PROGRAM Axis03_Command
VAR
//System_Bit
	Always_ON	:	BOOL	:=TRUE	;//상시 ON 
	Always_OFF	:	BOOL	:=FALSE	;//상시 OFF

//Motor_Command
	Axis03: AXIS_REF;											//Y축
	Axis03_MC_Power: MC_Power;
	Axis03_MC_Home: FB_HomeBeforeMoveAX8000;
	Axis03_Jog: MC_Jog;	
	Axis03_Home_Pos_Move: MC_MoveAbsolute;
	Axis03_Wait_Pos_Move: MC_MoveAbsolute;
	Axis03_Target_Pos_Move: MC_MoveAbsolute;
	Axis03_Work_End_Move: MC_MoveAbsolute;
	Axis03_Maint_Move: MC_MoveAbsolute;
	Axis03_Tool_Change: MC_MoveAbsolute;	
	Axis03_Calibration: MC_MoveAbsolute;	

	Timer02: TON;
END_VAR
VAR // added by the converter: edge detectors and wires of the graphical bodies
    _rt1, _rt2, _rt3 : R_TRIG;
END_VAR

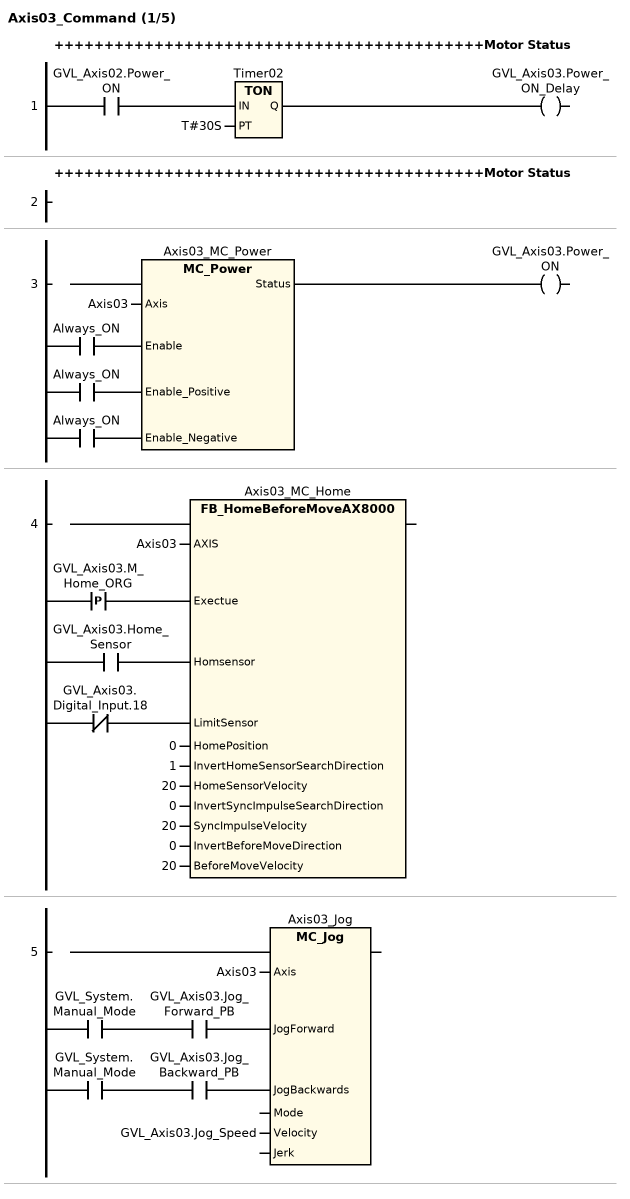
// NETWORK 1: +++++++++++++++++++++++++++++++++++++++++++Motor Status
Timer02(IN := GVL_Axis02.Power_ON, PT := T#30S); // TON
GVL_Axis03.Power_ON_Delay := Timer02.Q;

// NETWORK 2: +++++++++++++++++++++++++++++++++++++++++++Motor Status

// NETWORK 3
Axis03_MC_Power(
    Axis := Axis03,
    Enable := Always_ON,
    Enable_Positive := Always_ON,
    Enable_Negative := Always_ON); // MC_Power
GVL_Axis03.Power_ON := Axis03_MC_Power.Status;

// NETWORK 4
_rt1(CLK := GVL_Axis03.M_Home_ORG);
Axis03_MC_Home(
    AXIS := Axis03,
    Exectue := _rt1.Q,
    Homsensor := GVL_Axis03.Home_Sensor,
    LimitSensor := NOT GVL_Axis03.Digital_Input.18,
    HomePosition := 0,
    InvertHomeSensorSearchDirection := 1,
    HomeSensorVelocity := 20,
    InvertSyncImpulseSearchDirection := 0,
    SyncImpulseVelocity := 20,
    InvertBeforeMoveDirection := 0,
    BeforeMoveVelocity := 20); // FB_HomeBeforeMoveAX8000

// NETWORK 5
Axis03_Jog(
    Axis := Axis03,
    JogForward := GVL_System.Manual_Mode AND GVL_Axis03.Jog_Forward_PB,
    JogBackwards := GVL_System.Manual_Mode AND GVL_Axis03.Jog_Backward_PB,
    Velocity := GVL_Axis03.Jog_Speed); // MC_Jog

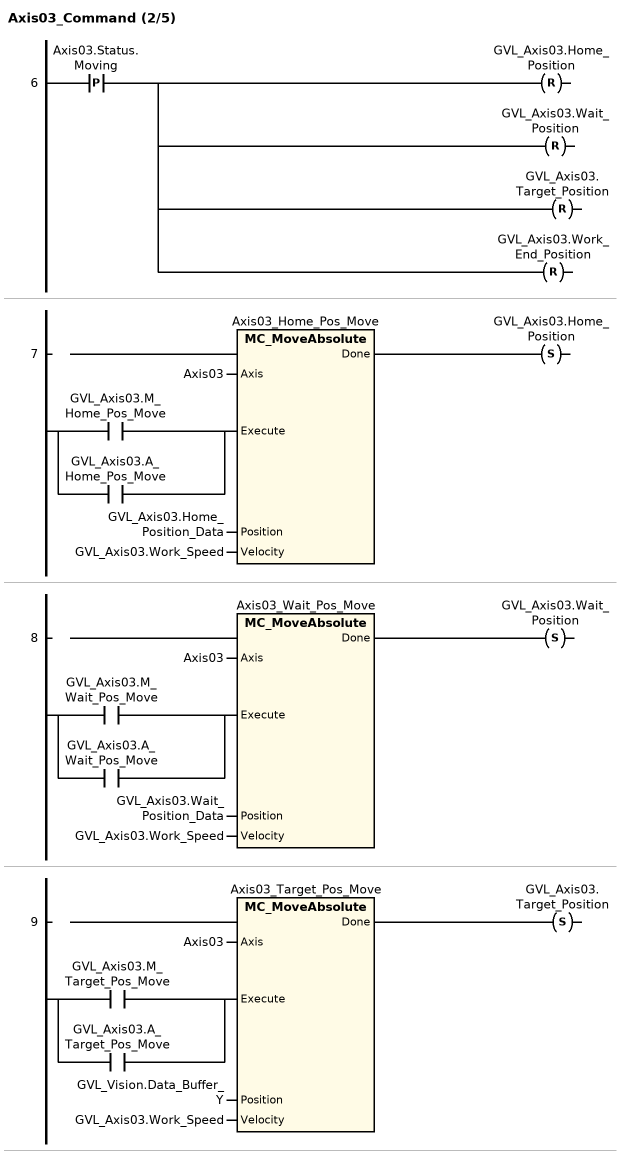
// NETWORK 6
_rt2(CLK := Axis03.Status.Moving);
GVL_Axis03.Home_Position R= _rt2.Q;
GVL_Axis03.Wait_Position R= _rt2.Q;
GVL_Axis03.Target_Position R= _rt2.Q;
GVL_Axis03.Work_End_Position R= _rt2.Q;

// NETWORK 7
Axis03_Home_Pos_Move(
    Axis := Axis03,
    Execute := GVL_Axis03.M_Home_Pos_Move OR GVL_Axis03.A_Home_Pos_Move,
    Position := GVL_Axis03.Home_Position_Data,
    Velocity := GVL_Axis03.Work_Speed); // MC_MoveAbsolute
GVL_Axis03.Home_Position S= Axis03_Home_Pos_Move.Done;

// NETWORK 8
Axis03_Wait_Pos_Move(
    Axis := Axis03,
    Execute := GVL_Axis03.M_Wait_Pos_Move OR GVL_Axis03.A_Wait_Pos_Move,
    Position := GVL_Axis03.Wait_Position_Data,
    Velocity := GVL_Axis03.Work_Speed); // MC_MoveAbsolute
GVL_Axis03.Wait_Position S= Axis03_Wait_Pos_Move.Done;

// NETWORK 9
Axis03_Target_Pos_Move(
    Axis := Axis03,
    Execute := GVL_Axis03.M_Target_Pos_Move OR GVL_Axis03.A_Target_Pos_Move,
    Position := GVL_Vision.Data_Buffer_Y,
    Velocity := GVL_Axis03.Work_Speed); // MC_MoveAbsolute
GVL_Axis03.Target_Position S= Axis03_Target_Pos_Move.Done;

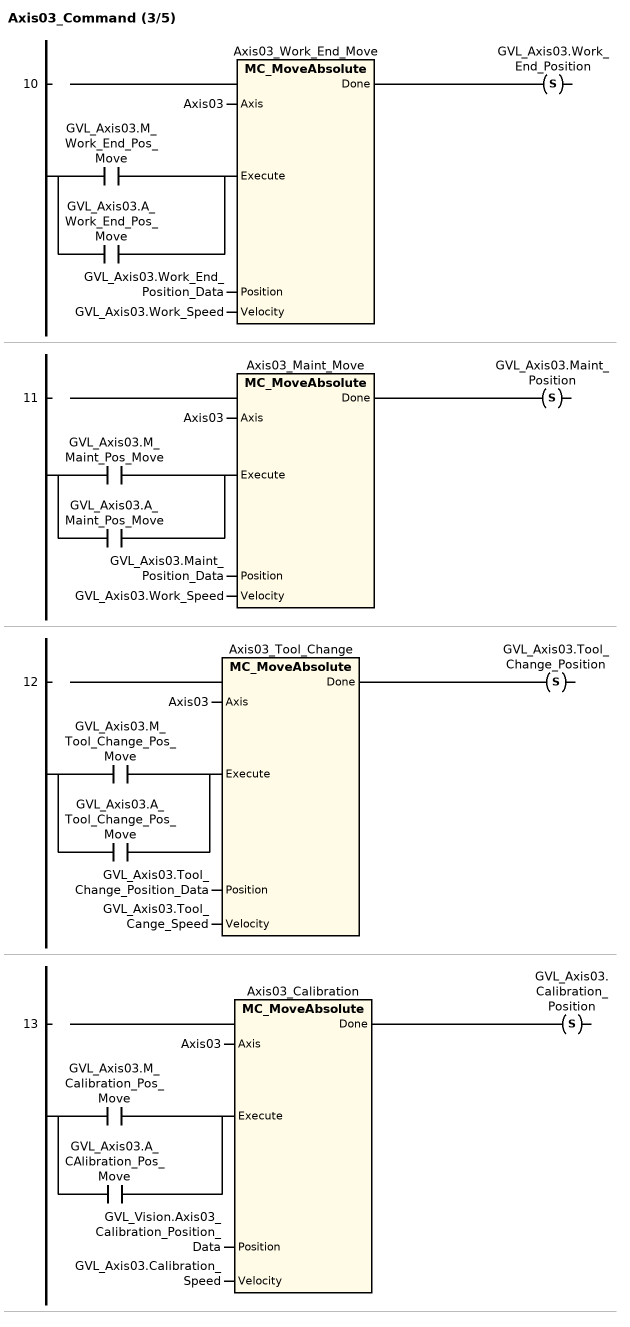
// NETWORK 10
Axis03_Work_End_Move(
    Axis := Axis03,
    Execute := GVL_Axis03.M_Work_End_Pos_Move OR GVL_Axis03.A_Work_End_Pos_Move,
    Position := GVL_Axis03.Work_End_Position_Data,
    Velocity := GVL_Axis03.Work_Speed); // MC_MoveAbsolute
GVL_Axis03.Work_End_Position S= Axis03_Work_End_Move.Done;

// NETWORK 11
Axis03_Maint_Move(
    Axis := Axis03,
    Execute := GVL_Axis03.M_Maint_Pos_Move OR GVL_Axis03.A_Maint_Pos_Move,
    Position := GVL_Axis03.Maint_Position_Data,
    Velocity := GVL_Axis03.Work_Speed); // MC_MoveAbsolute
GVL_Axis03.Maint_Position S= Axis03_Maint_Move.Done;

// NETWORK 12
Axis03_Tool_Change(
    Axis := Axis03,
    Execute := GVL_Axis03.M_Tool_Change_Pos_Move OR GVL_Axis03.A_Tool_Change_Pos_Move,
    Position := GVL_Axis03.Tool_Change_Position_Data,
    Velocity := GVL_Axis03.Tool_Cange_Speed); // MC_MoveAbsolute
GVL_Axis03.Tool_Change_Position S= Axis03_Tool_Change.Done;

// NETWORK 13
Axis03_Calibration(
    Axis := Axis03,
    Execute := GVL_Axis03.M_Calibration_Pos_Move OR GVL_Axis03.A_CAlibration_Pos_Move,
    Position := GVL_Vision.Axis03_Calibration_Position_Data,
    Velocity := GVL_Axis03.Calibration_Speed); // MC_MoveAbsolute
GVL_Axis03.Calibration_Position S= Axis03_Calibration.Done;

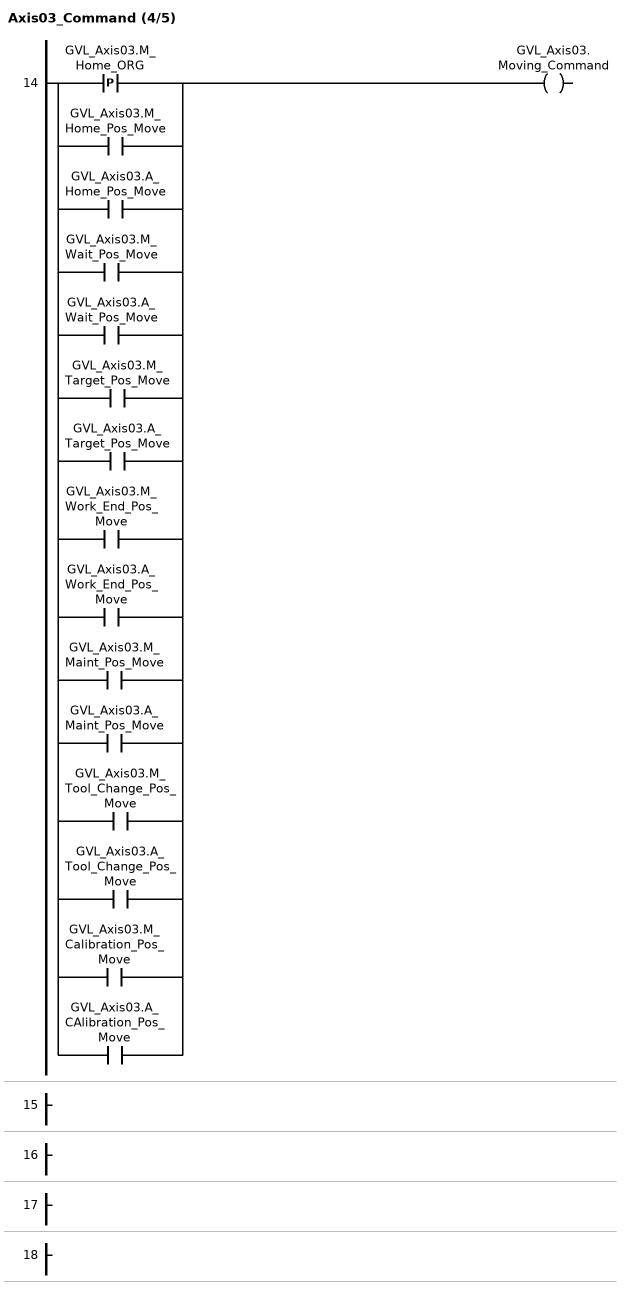
// NETWORK 14
_rt3(CLK := GVL_Axis03.M_Home_ORG);
GVL_Axis03.Moving_Command := _rt3.Q OR GVL_Axis03.M_Home_Pos_Move OR GVL_Axis03.A_Home_Pos_Move OR GVL_Axis03.M_Wait_Pos_Move OR GVL_Axis03.A_Wait_Pos_Move OR GVL_Axis03.M_Target_Pos_Move OR GVL_Axis03.A_Target_Pos_Move OR GVL_Axis03.M_Work_End_Pos_Move OR GVL_Axis03.A_Work_End_Pos_Move OR GVL_Axis03.M_Maint_Pos_Move OR GVL_Axis03.A_Maint_Pos_Move OR GVL_Axis03.M_Tool_Change_Pos_Move OR GVL_Axis03.A_Tool_Change_Pos_Move OR GVL_Axis03.M_Calibration_Pos_Move OR GVL_Axis03.A_CAlibration_Pos_Move;

// NETWORK 15

// NETWORK 16

// NETWORK 17

// NETWORK 18

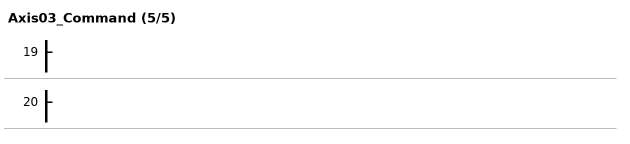
// NETWORK 19

// NETWORK 20

END_PROGRAM

(* stored: Version 1.1.0.1, ProductVersion 3.1.4024.15
   POU Axis03_Command: Id {2dae8a82-6a5e-4e7f-8d3f-803907bc122f}, SpecialFunc None *)
